Yaskawa INFORM job: R1_W72(-45,-90)R2.JBI

/JOB
//NAME R1_W72(-45,-90)R2
///FOLDERNAME KRIS-SCIANA
//POS
///NPOS 47,47,0,3,0,0
///TOOL 0
///POSTYPE PULSE
///PULSE
C00000=-2935,-133602,-129570,-25637,29822,84022
C00001=107670,22375,-20897,-3217,90322,-84959
C00002=107670,17970,6436,-3368,71268,-84460
C00003=107652,18775,11341,-3415,68666,-84393
C00004=107423,16216,11848,-3383,67035,-84428
C00005=107510,17738,13983,-3423,66508,-84381
C00006=107644,19198,13406,-3437,67615,-84365
C00007=105864,18950,14991,-2899,66440,-84981
C00008=105786,18051,14668,-2879,66175,-85004
C00009=107638,19551,14976,-3454,66830,-84344
C00010=107646,19083,12865,-3431,67888,-84372
C00011=107665,17340,-1125,-3297,75589,-84580
C00012=111696,-2239,-29974,-4412,83454,80233
C00013=107330,14705,-3413,-3195,75631,79014
C00014=107228,13360,-2084,-3185,74119,79019
C00015=107298,14404,-556,-3212,73719,79054
C00016=107330,14766,-1706,-3209,74613,79041
C00017=107372,15462,-55,-3230,73955,79074
C00018=107289,14311,-411,-3211,73580,79055
C00019=107329,14769,-1561,-3210,74526,79043
C00020=107333,14883,-471,-3220,73914,79061
C00021=107047,14897,3200,-3167,71654,79019
C00022=106435,14835,3634,-2983,71333,78810
C00023=107333,15238,3155,-3253,71868,79115
C00024=107330,14705,-3413,-3195,75631,79014
C00025=100153,28277,550,-5705,79007,75993
C00026=100153,27887,7605,-5801,74487,76204
C00027=107285,22854,7276,-8115,72731,78794
C00028=107334,22018,6550,-8130,72754,78811
C00029=107440,25166,9559,-8172,72533,78863
C00030=107226,20659,5973,-8992,71673,77785
C00031=107013,14456,2681,-11673,68462,74803
C00032=107194,14536,2804,-11739,68452,74869
C00033=107272,14744,5152,-11872,67155,75033
C00034=109703,9347,4240,-12926,65365,76135
C00035=107337,14954,-210,-12591,69921,73644
C00036=112500,13425,-9878,-17180,79722,-74576
C00037=112485,14733,7938,-17950,69883,-73131
C00038=111969,16057,13283,-18104,67283,-72919
C00039=110684,15822,14890,-17875,65942,-73199
C00040=111800,14785,12888,-18108,66854,-72915
C00041=111841,17958,15807,-18141,66705,-72876
C00042=106114,15731,9225,-16109,68282,-75285
C00043=107338,15945,7393,-16354,69717,-75029
C00044=107338,15248,2657,-16122,72176,-75369
C00045=107337,19186,-22088,-15454,88814,-77512
C00046=19636,17486,-23676,-16883,89789,-76092
BC00000=155306,23208,1075173
BC00001=10055,561207,1075175
BC00002=10055,561207,1075175
BC00003=10767,561196,1075175
BC00004=11308,559778,1075175
BC00005=11308,559778,1075175
BC00006=11053,561191,1075175
BC00007=11110,561431,1075175
BC00008=11110,561431,1075175
BC00009=11110,561431,1075175
BC00010=10825,561435,1075175
BC00011=10112,561447,1075175
BC00012=140937,561120,1075175
BC00013=141696,561154,1075175
BC00014=142236,559895,1075175
BC00015=142236,559895,1075175
BC00016=141999,561168,1075175
BC00017=143361,561968,1075175
BC00018=143361,561968,1075175
BC00019=143340,560337,1075175
BC00020=126626,559274,1075175
BC00021=126734,565078,1075175
BC00022=126734,565078,1075175
BC00023=126734,565078,1075175
BC00024=141696,561154,1075175
BC00025=128122,568868,1075175
BC00026=128122,568868,1075175
BC00027=155211,570997,1075175
BC00028=129858,568975,1075175
BC00029=129858,568975,1075175
BC00030=147054,569224,1075175
BC00031=122568,563903,1075175
BC00032=122568,563903,1075175
BC00033=113555,566058,1075175
BC00034=113554,566057,1075171
BC00035=107709,567124,1075175
BC00036=15,555872,1075175
BC00037=15,555877,1075175
BC00038=15,555966,1075175
BC00039=15,556001,1075175
BC00040=15,556001,1075175
BC00041=15,556001,1075175
BC00042=99510,564948,1075175
BC00043=101317,565127,1075175
BC00044=99872,565038,1075175
BC00045=99830,565033,1075175
BC00046=99830,7321,1075175
///POSTYPE BASE
///RECTAN
///RCONF 0,0,0,0,1,0,0,0,0,0,0,0,0,0,0,0,0,0,0,0,0,0,0,0
P00006=2.006,1.622,-0.565,0.0000,0.0000,0.0000
P00021=0.073,2.058,-0.109,0.0000,0.0000,0.0000
P00022=2.006,1.622,-0.565,0.0000,0.0000,0.0000
//INST
///DATE 2024/09/12 13:43
///ATTR SC,RW
///GROUP1 RB1,BS1
NOP
SFTOF
MOVJ C00000 BC00000 VJ=100.00
MOVJ C00001 BC00001 VJ=100.00
MOVJ C00002 BC00002 VJ=100.00
MOVL C00003 BC00003 V=100.0
MOVL C00004 BC00004 V=60.0
REFP 3 C00005 BC00005
CALL JOB:SEARCH-R1
SET P022 P006
SFTON P022
MOVL C00006 BC00006 V=60.0
MOVL C00007 BC00007 V=60.0
REFP 3 C00008 BC00008
CALL JOB:SEARCH-R1
SET P022 P006
SFTON P022
MOVL C00009 BC00009 V=60.0
MOVL C00010 BC00010 V=100.0
MOVJ C00011 BC00011 VJ=100.00
'Path S813
SFTOF
MOVJ C00012 BC00012 VJ=100.00
MOVL C00013 BC00013 V=100.0
MOVL C00014 BC00014 V=60.0
REFP 3 C00015 BC00015
CALL JOB:SEARCH-R1
SET P021 P006
SFTON P021
MOVL C00016 BC00016 V=60.0
MOVL C00017 BC00017 V=60.0
REFP 3 C00018 BC00018
CALL JOB:SEARCH-R1
SET P021 P006
SFTON P021
MOVL C00019 BC00019 V=60.0
MOVL C00020 BC00020 V=100.0
MOVL C00021 BC00021 V=60.0
REFP 3 C00022 BC00022
CALL JOB:SEARCH-R1
SET P021 P006
SFTON P021
MOVL C00023 BC00023 V=60.0
MOVL C00024 BC00024 V=166.7
'Path W108
SFTOF
SFTON P021
MOVJ C00025 BC00025 VJ=100.00
MOVL C00026 BC00026 V=100.0
CALL JOB:COFNIJ_DRUT
MACRO1 MJ#(0) ARGF6
MOVL C00027 BC00027 V=100.0 PL=0
REFP 1 C00028 BC00028
REFP 2 C00029 BC00029
ARCON
MOVL C00030 BC00030 V=10.0
MACRO1 MJ#(0) ARGF7
MOVL C00031 BC00031 V=10.8
MOVL C00032 BC00032 V=10.8
MOVL C00033 BC00033 V=10.8
MOVL C00034 BC00034 V=10.8
ARCOF
MOVL C00035 BC00035 V=166.7
SFTOF
'Path W110
SFTOF
SFTON P022
MOVJ C00036 BC00036 VJ=100.00
MOVJ C00037 BC00037 VJ=100.00
MOVL C00038 BC00038 V=100.0
MOVL C00039 BC00039 V=100.0 PL=0
REFP 1 C00040 BC00040
REFP 2 C00041 BC00041
MACRO1 MJ#(0) ARGF9
ARCON
SFTON P021
MOVL C00042 BC00042 V=10.8
ARCOF
MOVL C00043 BC00043 V=100.0
MOVL C00044 BC00044 V=100.0
MOVL C00045 BC00045 V=166.7
SFTOF
MOVJ C00046 BC00046 VJ=100.00
END
